PROGRAM P_DelayedLight_Test_CFC
VAR
	fbDelayedLight		:	FB_DelayedLight;
	bOn					:	BOOL;
	bOff				:	BOOL;
	bControlLevel		:	BOOL;
END_VAR

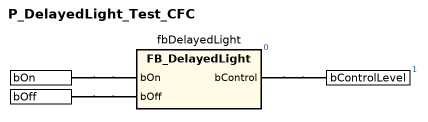
fbDelayedLight(bOn := bOn, bOff := bOff); // FB_DelayedLight
bControlLevel := fbDelayedLight.bControl;

END_PROGRAM

(* stored: Version 1.1.0.1, ProductVersion 3.1.4024.12
   POU P_DelayedLight_Test_CFC: Id {5095a31f-897b-4169-abe3-542905efb1ea}, SpecialFunc None *)
